FUNCTION_BLOCK FB_PipelineInner
VAR_INPUT
    value : INT;
END_VAR
VAR_OUTPUT
    bError : BOOL;
END_VAR

// Inner raises an error for any negative input.
bError := value < 0;

END_FUNCTION_BLOCK

(* stored: Version 1.1.0.1
   POU FB_PipelineInner: Id {622fc4d7-c996-4c5b-9887-5d1f8552b65a}, SpecialFunc None *)
